{attribute 'qualified_only'}
VAR_GLOBAL CONSTANT
	MAX_INIT_LIST: INT := 64;
END_VAR

(* stored: Version 1.1.0.1, ProductVersion 3.1.4024.9
   GVL INITIALIZE: Id {f533b537-69ac-4c5e-baf9-a64ab2e12df5} *)
